# B&R Automation Studio project lab1_KRBO_03_22
Automation Studio 4.5.2.102

## Configuration Config1

### Hardware
```
4PP065_0571_P74 : 4PP065.0571-P74 v1.1.2.0
  Connector IF5:
    ActivateDevice = 1
    Mode = Manual
    InternetAddress = 10.0.1.10
    SubnetMask = 255.255.255.0
  ConfigurationID = labBR
  Simulation = 1
```

## Logical view

### Global.var
```iecst
VAR
	regulator : FB_Regulator;
	speed : REAL;
	counter : UINT;
	enable : BOOL;
	motor2 : FB_Motor;
	motor : FB_Motor;
	integrator : FB_Integrator;
END_VAR
```

### Library Logical/Libraries/Library

#### Library.fun
```iecst
{REDUND_ERROR} FUNCTION_BLOCK FB_Integrator (*TODO: Add your comment here*) (*$GROUP=User,$CAT=User,$GROUPICON=User.png,$CATICON=User.png*)
	VAR_INPUT
		in : {REDUND_UNREPLICABLE} REAL;
		dt : REAL;
	END_VAR
	VAR_OUTPUT
		out : {REDUND_UNREPLICABLE} REAL;
	END_VAR
	VAR
		prev_value : REAL;
	END_VAR
END_FUNCTION_BLOCK

{REDUND_ERROR} FUNCTION_BLOCK FB_Regulator (*TODO: Add your comment here*) (*$GROUP=User,$CAT=User,$GROUPICON=User.png,$CATICON=User.png*)
	VAR_INPUT
		e : {REDUND_UNREPLICABLE} REAL;
	END_VAR
	VAR
		dt : REAL;
	END_VAR
	VAR_OUTPUT
		u : {REDUND_UNREPLICABLE} REAL;
	END_VAR
	VAR
		k_p : {REDUND_UNREPLICABLE} REAL;
		k_i : {REDUND_UNREPLICABLE} REAL;
		integrator : {REDUND_UNREPLICABLE} FB_Integrator;
		iyOld : {REDUND_UNREPLICABLE} REAL;
		max_abs_value : {REDUND_UNREPLICABLE} REAL;
		last_sum : {REDUND_UNREPLICABLE} REAL;
		sum : {REDUND_UNREPLICABLE} REAL;
	END_VAR
END_FUNCTION_BLOCK

{REDUND_ERROR} FUNCTION_BLOCK FB_Motor (*TODO: Add your comment here*) (*$GROUP=User,$CAT=User,$GROUPICON=User.png,$CATICON=User.png*)
	VAR_INPUT
		u : REAL;
	END_VAR
	VAR
		dt : REAL;
	END_VAR
	VAR_OUTPUT
		w : REAL;
		phi : REAL;
	END_VAR
	VAR
		Tm : REAL;
		integrator : FB_Integrator;
		ke : REAL;
	END_VAR
END_FUNCTION_BLOCK
```

#### FB_Integrator.c
```c
#include <bur/plctypes.h>
#ifdef __cplusplus
	extern "C"
	{
#endif
	#include "Library.h"
#ifdef __cplusplus
	};
#endif
/* TODO: Add your comment here */
void FB_Integrator(struct FB_Integrator* inst)
{
	/*TODO: Add your code here*/
	inst->out = inst->dt * inst->in + inst->prev_value;
	inst->prev_value = inst->out;
}
```

#### FB_Motor.c
```c
#include <bur/plctypes.h>
#ifdef __cplusplus
	extern "C"
	{
#endif
	#include "Library.h"
#ifdef __cplusplus
	};
#endif
/* TODO: Add your comment here */
void FB_Motor(struct FB_Motor* inst)
{
	inst->integrator.dt = inst->dt;
	REAL a = inst->u / inst->ke - inst->w;
	REAL b = a / inst->Tm;

	inst->integrator.in = b;
	FB_Integrator(&inst->integrator);

	inst->w = inst->integrator.out;
}
```

#### FB_Regulator.c
```c
#include <bur/plctypes.h>
#ifdef __cplusplus
	extern "C"
	{
#endif
	#include "Library.h"
#ifdef __cplusplus
	};
#endif
/* TODO: Add your comment here */
void FB_Regulator(struct FB_Regulator* inst)
{
	inst->integrator.dt = inst->dt;

	REAL a = inst->e * inst->k_p;
	REAL b = inst->e * inst->k_i;

	a = a > inst->max_abs_value ? inst->max_abs_value : a;
	a = a < -inst->max_abs_value ? -inst->max_abs_value : a;

	inst->integrator.in = b + inst->last_sum;
	FB_Integrator(&inst->integrator);

	inst->sum = a + inst->integrator.out;
	inst->u = inst->sum;
	inst->u = inst->u > inst->max_abs_value ? inst->max_abs_value : inst->u;
	inst->u = inst->u < -inst->max_abs_value ? -inst->max_abs_value : inst->u;

	inst->last_sum = inst->u - inst->sum;
}
```

### Program Logical/Program

#### Cyclic.c
```c
#include <bur/plctypes.h>

#ifdef _DEFAULT_INCLUDES
	#include <AsDefault.h>
#endif

void _CYCLIC ProgramCyclic(void)
{
	if(enable)
	{
		if(counter == 1000)
		{
			speed = 60;
		}
		if(counter == 1100)
		{
			speed = 0;
			counter = 0;
		}
		counter = counter + 1;

		regulator.e = speed - motor.w;
		FB_Regulator(&regulator);

		motor.u = regulator.u;
		FB_Motor(&motor);

		motor2.u = speed * motor2.ke;
		FB_Motor(&motor2);
	}
}
```

#### Init.c
```c
#include <bur/plctypes.h>

#ifdef _DEFAULT_INCLUDES
	#include <AsDefault.h>
#endif

void _INIT ProgramInit(void)
{
	motor.dt = 0.02;
	motor.ke = 0.32;
	motor.Tm = 0.2;
	motor.u = 0;

	motor2.dt = 0.02;
	motor2.ke = 0.32;
	motor2.Tm = 0.2;
	motor2.u = 0;

	regulator.dt = 0.01;
	regulator.k_i = 4.3;
	regulator.k_p = 0.36;
	regulator.max_abs_value = 27.0;

	speed = 0;
	counter = 0;
	enable = 1;
}
```
